FUNCTION_BLOCK FB_PT100_10DIN_EL3202 IMPLEMENTS I_TemperatureSensor
VAR
//Temperature measurement: PT 100 1/10 DIN + EL3202:(0010,0020,0030) 4-wire
	//Propertie Real value
	fTemperature : REAL;
	//Raw value
	TempRaw AT %I* : INT;
	//Convertion parameters
	m : REAL := 0.01; //Multiplier for convertion
END_VAR

PROPERTY Temperature : REAL
GET
fTemperature := INT_TO_REAL(TempRaw) * m;
Temperature := THIS^.fTemperature;
END_GET
END_PROPERTY

END_FUNCTION_BLOCK

(* stored: Version 1.1.0.1
   POU FB_PT100_EL3202: Id {f24975da-7fc4-4f10-9889-9699ffa676d5}, SpecialFunc None
   Property Temperature: Id {b4f94d05-8b7b-4a89-bced-d4aeaf7c4cdd}
   Get Get: Id {3b760b93-52e2-4ec0-9e36-25f20554f12f} *)
